Yaskawa INFORM job: plata_tarpez_planes_program.JBI

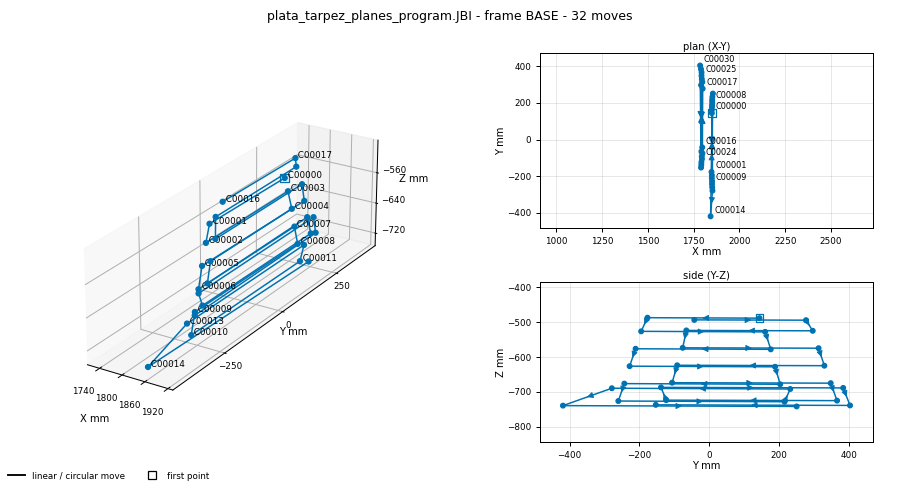
[picture p0: tool path of plata_tarpez_planes_program.JBI in frame BASE, 32 of 35 moves have a stored position in this frame; points joined in program order, loops and branches not executed]
/JOB
//NAME plata_tarpez_planes_program
//POS
///NPOS 32,0,32,0,0,0
///TOOL 0
///POSTYPE BASE
///RECTAN
///RCONF 0,0,0,0,0,0,0,0,0,0,0,0,0,0,0,0,0,0,0,0,0,0,0,0
C00000=1849.133670,144.284796,-488.447771,5.000000,-87.635501,175.000000
C00001=1847.396284,-176.926772,-487.144143,5.000000,-87.635501,175.000000
C00002=1849.267966,-195.060780,-526.264765,5.000000,-87.635501,175.000000
C00003=1848.597057,160.509809,-527.814951,5.000000,-87.635501,175.000000
C00004=1850.040996,176.550291,-577.867075,5.000000,-87.635501,175.000000
C00005=1849.002120,-211.010003,-576.250515,5.000000,-87.635501,175.000000
C00006=1850.295485,-228.153559,-626.166769,5.000000,-87.635501,175.000000
C00007=1850.505582,188.891524,-627.943799,5.000000,-87.635501,175.000000
C00008=1851.287857,203.613283,-678.017598,5.000000,-87.635501,175.000000
C00009=1850.058174,-243.308589,-676.154742,5.000000,-87.635501,175.000000
C00010=1851.133087,-260.546627,-726.079611,5.000000,-87.635501,175.000000
C00011=1851.024678,216.067379,-728.124855,5.000000,-87.635501,175.000000
C00012=1851.987053,232.428968,-691.595698,5.000000,-87.635501,175.000000
C00013=1852.519718,-279.090275,-689.383479,5.000000,-87.635501,175.000000
C00014=1842.199338,-419.244640,-739.252572,5.000000,-87.635501,175.000000
C00015=1854.725679,250.752364,-741.604138,180.000000,-60.000000,0.000000
C00016=1796.676954,-42.745927,-493.412027,-5.000000,-88.422259,175.000000
C00017=1799.034185,277.636243,-494.253813,-5.000000,-88.422259,175.000000
C00018=1790.412920,296.914300,-524.731128,-5.000000,-88.422259,175.000000
C00019=1792.148212,-65.518147,-523.657612,-5.000000,-88.422259,175.000000
C00020=1797.807056,-75.873201,-573.491602,-5.000000,-88.422259,175.000000
C00021=1797.122597,313.677206,-574.612921,-5.000000,-88.422259,175.000000
C00022=1794.429068,330.248363,-624.753172,-5.000000,-88.422259,175.000000
C00023=1794.321675,-91.724515,-623.561906,-5.000000,-88.422259,175.000000
C00024=1795.070152,-106.337756,-673.519096,-5.000000,-88.422259,175.000000
C00025=1792.725845,348.444906,-674.870747,-5.000000,-88.422259,175.000000
C00026=1793.013084,366.616758,-724.933427,-5.000000,-88.422259,175.000000
C00027=1792.213640,-123.206976,-723.569198,-5.000000,-88.422259,175.000000
C00028=1791.552170,-138.180900,-686.961662,-5.000000,-88.422259,175.000000
C00029=1789.938232,384.250698,-688.484649,-5.000000,-88.422259,175.000000
C00030=1785.273624,403.858246,-738.687785,-5.000000,-88.422259,175.000000
C00031=1790.286080,-153.093012,-736.973496,180.000000,-60.000000,0.000000
///POSTYPE PULSE
///PULSE
EC00000=172032.0
EC00001=172032.0
EC00002=172032.0
EC00003=172032.0
EC00004=172032.0
EC00005=172032.0
EC00006=172032.0
EC00007=172032.0
EC00008=172032.0
EC00009=172032.0
EC00010=172032.0
EC00011=172032.0
EC00012=172032.0
EC00013=172032.0
EC00014=172032.0
EC00015=172032.0
EC00016=356352.0
EC00017=356352.0
EC00018=356352.0
EC00019=356352.0
EC00020=356352.0
EC00021=356352.0
EC00022=356352.0
EC00023=356352.0
EC00024=356352.0
EC00025=356352.0
EC00026=356352.0
EC00027=356352.0
EC00028=356352.0
EC00029=356352.0
EC00030=356352.0
EC00031=356352.0
//INST
///DATE 2023/08/16 14:07
///ATTR SC,RW,RJ
////FRAME BASE
///GROUP1 RB1,ST1
NOP
MOVJ P009 EX000 VJ=15.00
MOVJ C00000 EC00000 VJ=15.0
CALL JOB:SPYON
MOVL C00001 EC00001 V=150.0
MOVL C00002 EC00002 V=150.0
MOVL C00003 EC00003 V=150.0
MOVL C00004 EC00004 V=150.0
MOVL C00005 EC00005 V=150.0
MOVL C00006 EC00006 V=150.0
MOVL C00007 EC00007 V=150.0
MOVL C00008 EC00008 V=150.0
MOVL C00009 EC00009 V=150.0
MOVL C00010 EC00010 V=150.0
MOVL C00011 EC00011 V=150.0
MOVL C00012 EC00012 V=150.0
MOVL C00013 EC00013 V=150.0
MOVL C00014 EC00014 V=150.0
MOVL C00015 EC00015 V=150.0
CALL JOB:SPYOF
MOVJ P009 VJ=15.00
MOVJ C00016 EC00016 VJ=15.0
CALL JOB:SPYON
MOVL C00017 EC00017 V=150.0
MOVL C00018 EC00018 V=150.0
MOVL C00019 EC00019 V=150.0
MOVL C00020 EC00020 V=150.0
MOVL C00021 EC00021 V=150.0
MOVL C00022 EC00022 V=150.0
MOVL C00023 EC00023 V=150.0
MOVL C00024 EC00024 V=150.0
MOVL C00025 EC00025 V=150.0
MOVL C00026 EC00026 V=150.0
MOVL C00027 EC00027 V=150.0
MOVL C00028 EC00028 V=150.0
MOVL C00029 EC00029 V=150.0
MOVL C00030 EC00030 V=150.0
MOVL C00031 EC00031 V=150.0
CALL JOB:SPYOF
MOVJ P009 VJ=15.00
END
